// TIA Portal V17 export
// export: Created 2023-02-22T17:45:26.1519381Z, ExportSetting WithDefaults, DisplayName Totally Integrated Automation Portal, DisplayVersion V17, DisplayName TIA Portal Openness, DisplayVersion V17, DisplayName TIA Portal Version Control Interface, DisplayVersion V17, DisplayName TIA Portal Test Suite Advanced, DisplayVersion V17, DisplayName STEP 7 Professional, DisplayVersion V17, DisplayName SIMATIC Energy Suite, DisplayVersion V17, DisplayName STEP 7 Safety, DisplayVersion V17, DisplayName WinCC Professional, DisplayVersion V17
FUNCTION "MAN_ChooseMode" : Void   // FC7, LAD
{ S7_Optimized_Access := 'TRUE' }
VERSION : 0.1
// stored: AutoNumber true, IsIECCheckEnabled false, SetENOAutomatically false, UDAEnableTagReadback false
   VAR_INPUT
      ButtonAuto : Bool;
      ButtonManual : Bool;
   END_VAR
   VAR_OUTPUT
      Auto : Bool;
      Manual : Bool;
   END_VAR
BEGIN

REGION Network 1
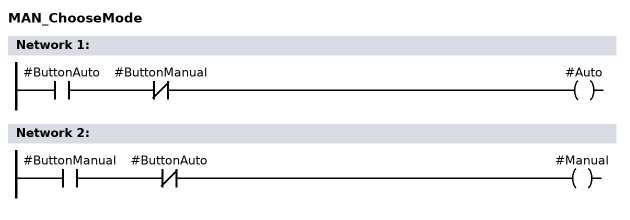
   RUNG wire#powerrail
      Contact( #ButtonAuto )
      I_Contact( #ButtonManual )
      Coil( #Auto )
   END_RUNG
   // the same network as SCL:
   #Auto := #ButtonAuto AND NOT #ButtonManual;
END_REGION

REGION Network 2
   RUNG wire#powerrail
      Contact( #ButtonManual )
      I_Contact( #ButtonAuto )
      Coil( #Manual )
   END_RUNG
   // the same network as SCL:
   #Manual := #ButtonManual AND NOT #ButtonAuto;
END_REGION
END_FUNCTION
